{attribute 'qualified_only'}
VAR_GLOBAL
	{attribute 'OPC.UA.DA' := '1'}
	{attribute 'OPC.UA.DA.Access' := '1'}
	{attribute 'init_namespace'} 
	Name : STRING(255);	
END_VAR

(* stored: Version 1.1.0.1
   GVL CurrentNamespace: Id {7ab8fe4a-b63a-03ec-3a27-3dabf7754d3b} *)
